ABB RobotStudio station: Solution_final_v2.rsstn

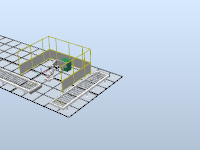
Station Solution1_1 (saved by RobotStudio 21.1.9393.1)
Controller Controlador1, task T_ROB1: task frame (RAPID world) sits at (-200, -1000, 0) mm in the station
Controller Controlador1
  mechanical unit ROB_1: IRB1600_6_120__02, 6 joints, base frame (0, 0, 0) mm
Layout (positions relative to the parent item):
  - IRB1600_6_120__02 [mechanism, from Robots\IRB1600_6_120_G_02.rslib] at (-200, -1000, 0) mm; joint values [0.1941, 0.1473, -0.2355, 0.1043, 1.3308, 0.4277] (rad or m)
  - RA_MTG4000_22 [mechanism, from Tools\Fronius_Robacta_MTG4000_22deg.rslib] at (621.28, -831.87, 948.02) mm, rotated rx 166.41 ry 14.43 rz 164.42 deg
  - Fence_740 [graphiccomponentgroup, from Equipment\Fence_740.rslib] at (2000, 225, 0) mm
    - Body 1 [part, from Equipment\Fence_740.rslib]
    - Body 2 [part, from Equipment\Fence_740.rslib]
  - Fence_740_2 [graphiccomponentgroup, from Equipment\Fence_740.rslib] at (2000, 925, 0) mm, rotated rx 0 ry 0 rz 90 deg
    - Body 1 [part, from Equipment\Fence_740.rslib]
    - Body 2 [part, from Equipment\Fence_740.rslib]
  - Fence_740_3 [graphiccomponentgroup, from Equipment\Fence_740.rslib] at (2000, -2940, 0) mm, rotated rx 0 ry 0 rz 90 deg
    - Body 1 [part, from Equipment\Fence_740.rslib]
    - Body 2 [part, from Equipment\Fence_740.rslib]
  - Fence_740_4 [graphiccomponentgroup, from Equipment\Fence_740.rslib] at (2000, -2240, 0) mm, rotated rx 0 ry 0 rz 180 deg
    - Body 1 [part, from Equipment\Fence_740.rslib]
    - Body 2 [part, from Equipment\Fence_740.rslib]
  - Fence_2500 [graphiccomponentgroup, from Equipment\Fence_2500.rslib] at (2000, 225, 0) mm, rotated rx 0 ry 0 rz 180 deg
    - Body 1 [part, from Equipment\Fence_2500.rslib]
    - Body 2 [part, from Equipment\Fence_2500.rslib]
  - Fence_2500_2 [graphiccomponentgroup, from Equipment\Fence_2500.rslib] at (1300, 925, 0) mm, rotated rx 0 ry 0 rz 90 deg
    - Body 1 [part, from Equipment\Fence_2500.rslib]
    - Body 2 [part, from Equipment\Fence_2500.rslib]
  - Fence_2500_3 [graphiccomponentgroup, from Equipment\Fence_2500.rslib] at (1300, -2940, 0) mm, rotated rx 0 ry 0 rz 90 deg
    - Body 1 [part, from Equipment\Fence_2500.rslib]
    - Body 2 [part, from Equipment\Fence_2500.rslib]
  - ConveyorControl_2 [smart component, from Components\ConveyorControl.rslib]
      properties: Conveyor=(none)
  - Process [smart component]
      signals: DI inicio, DI inicio2, DO sal_conv1, DO sal_conv2
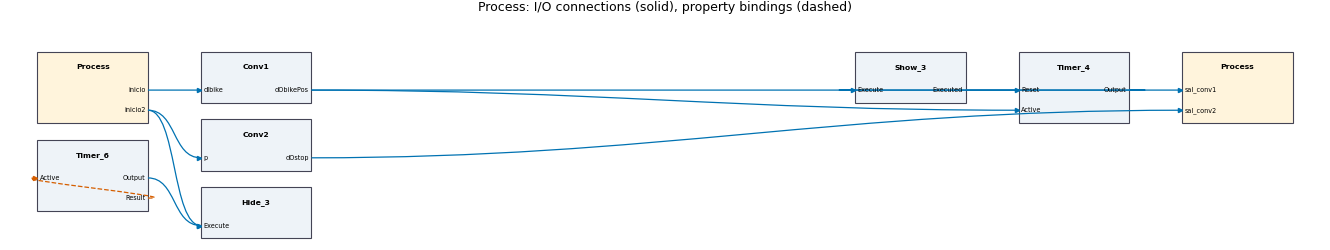
      connections:
        Timer_4.Output -> Show_3.Execute
        Show_3.Executed -> Timer_4.Reset
        Process.inicio -> Conv1.dIbike
        Conv1.dObikePos -> Timer_4.Active
        Timer_6.Output -> Hide_3.Execute
        Process.inicio2 -> Hide_3.Execute
        Conv1.dObikePos -> Process.sal_conv1
        Process.inicio2 -> Conv2.p
        Conv2.dOstop -> Process.sal_conv2
        Expression.Result => Timer_6.Active
    - Show_3 [smart component, from Components\Show.rslib]
        properties: Object=Bicycle Frame:1
    - Conv1 [smart component]
        signals: DI dIbike, DO dObikePos
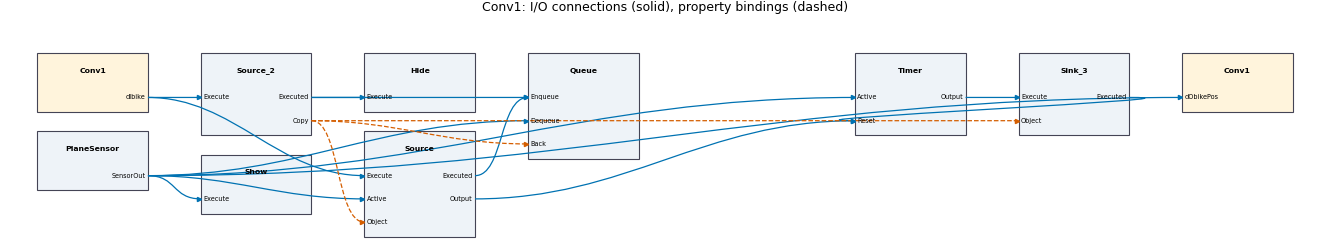
        connections:
          Conv1.dIbike -> Source.Execute
          Source.Executed -> Queue.Enqueue
          Conv1.dIbike -> Source_2.Execute
          Source_2.Executed -> Queue.Enqueue
          PlaneSensor.SensorOut -> Queue.Dequeue
          Source_2.Executed -> Hide.Execute
          PlaneSensor.SensorOut -> Show.Execute
          PlaneSensor.SensorOut -> Timer.Active
          Timer.Output -> Sink_3.Execute
          PlaneSensor.SensorOut -> Timer_5.Active
          Timer_5.Output -> Timer.Reset
          Sink_3.Executed -> Timer.Reset
          PlaneSensor.SensorOut -> Conv1.dObikePos
          Source_2.Copy => Queue.Back
          Source_2.Copy => Sink_2.Object
          Source_2.Copy => Sink_3.Object
      - 950_4800_h2 [part, from Equipment\Conveyor 950 4800 h2.rslib] at (2000, -3500, 0) mm, rotated rx 0 ry 0 rz 180 deg
      - Queue [smart component, from Components\Queue.rslib]
          properties: Back=(none); Front=(none); Queue={da4324a3-2cbe-466d-a78a-5e31958a6c5f};{e6e05bde-ee74-4659-88fe-c98839943faa};{f81fb27c-e148-4b64-9271-b941438183ca};{ce758764-b67b-4225-94dd-49e0e7ae394e}; NumberOfObjects=0
      - LinearMover [smart component, from Components\LinearMover.rslib]
          properties: Object=Queue; Direction=[-1 0 0]; Speed=0.5; Reference=Global; ReferenceObject=(none)
      - PlaneSensor [smart component, from Components\PlaneSensor.rslib]
          properties: Origin=[-2.65992 -3.5 0.435]; Axis1=[0 -0.91 0]; Axis2=[0 0 0.2]; SensedPart=(none)
        - _sensorPart_ [part]
      - Source_2 [smart component, from Components\Source.rslib]
          properties: Source=Bike; Copy=(none); Parent=(none); Position=[0 0 0]; Orientation=[0 0 0]; Transient=false; PhysicsBehavior=0
      - Show [smart component, from Components\Show.rslib]
          properties: Object=Bike
      - Hide [smart component, from Components\Hide.rslib]
          properties: Object=Bike
      - Sink_3 [smart component, from Components\Sink.rslib]
          properties: Object=(none)
      - Timer [smart component, from Components\Timer.rslib]
          properties: StartTime=3; Interval=3; Repeat=false; CurrentTime=0
    - Timer_4 [smart component, from Components\Timer.rslib]
        properties: StartTime=3; Interval=3; Repeat=false; CurrentTime=0
    - Conv2 [smart component]
        signals: DI p, DO dOstop
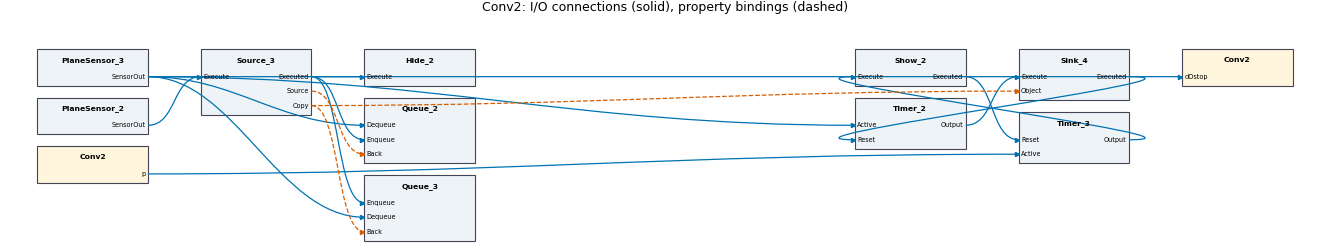
        connections:
          PlaneSensor_3.SensorOut -> Queue_2.Dequeue
          Source_3.Executed -> Queue_2.Enqueue
          Source_3.Executed -> Queue_3.Enqueue
          PlaneSensor_3.SensorOut -> Queue_3.Dequeue
          Source_3.Executed -> Hide_2.Execute
          PlaneSensor_3.SensorOut -> Timer_2.Active
          Timer_2.Output -> Sink_4.Execute
          Sink_4.Executed -> Timer_2.Reset
          PlaneSensor_2.SensorOut -> Source_3.Execute
          Timer_3.Output -> Show_2.Execute
          Show_2.Executed -> Timer_3.Reset
          Conv2.p -> Timer_3.Active
          PlaneSensor_3.SensorOut -> Conv2.dOstop
          Source_3.Source => Queue_2.Back
          Source_3.Copy => Queue_3.Back
          Source_3.Copy => Sink_4.Object
      - 950_4800_h2_3 [part, from Equipment\Conveyor 950 4800 h2.rslib] at (-1700, -1500, 0) mm, rotated rx 0 ry 0 rz 90 deg
      - Source_3 [smart component, from Components\Source.rslib]
          properties: Source=Bike2; Copy=Bike2_46; Parent=(none); Position=[0 0 0]; Orientation=[0 0 0]; Transient=false; PhysicsBehavior=0
      - LinearMover_2 [smart component, from Components\LinearMover.rslib]
          properties: Object=Queue_3; Direction=[0 1 0]; Speed=0.5; Reference=Global; ReferenceObject=(none)
      - PlaneSensor_2 [smart component, from Components\PlaneSensor.rslib]
          properties: Origin=[-2.61 -1.247316 0.435]; Axis1=[0.91 0 0]; Axis2=[0 0 0.2]; SensedPart=(none)
        - _sensorPart_ [part]
      - PlaneSensor_3 [smart component, from Components\PlaneSensor.rslib]
          properties: Origin=[-2.61 3.153624 0.435]; Axis1=[0.91 0 0]; Axis2=[0 0 0.2]; SensedPart=(none)
        - _sensorPart_ [part]
      - Hide_2 [smart component, from Components\Hide.rslib]
          properties: Object=Bike2
      - Show_2 [smart component, from Components\Show.rslib]
          properties: Object=Bike2
      - Queue_3 [smart component, from Components\Queue.rslib]
          properties: Back=Bike2_46; Front=Bike2_46; Queue={1f08c73b-8c5d-47c5-8fad-b47ddc3f47b2};{69fdafc0-c70e-498c-bd5d-4343ecce45a8};{ab0811c3-1ba0-43c0-b674-f4a10a17c4ae};{44498bd1-b295-4fc8-a058-8143949b90d9};{61c4f5f8-9c20-4886-aed5-0f792fba9fef};{207447c9-6041-471c-927b-d307d36bb852};{d11dc4f1-6705-4b2f-9a87-b3149d9034c5};{ffd23da9-bf60-4005-aac2-4753273c3d85};{c9eaf6c6-1d88-4ec3-ab1c-7dd69f2dac15}; NumberOfObjects=1
      - Sink_4 [smart component, from Components\Sink.rslib]
          properties: Object=Bike2_46
      - Timer_2 [smart component, from Components\Timer.rslib]
          properties: StartTime=3; Interval=3; Repeat=false; CurrentTime=0
      - Timer_3 [smart component, from Components\Timer.rslib]
          properties: StartTime=3; Interval=3; Repeat=true; CurrentTime=0
    - Hide_3 [smart component, from Components\Hide.rslib]
        properties: Object=Bicycle Frame:1
  - Bike [part]
  - Bike2 [part]
  - Soporte [smart component]
      signals: DI in_sop1, DI in_sop2, DI in_sop3, DO out_sop1, DO out_sop2, DO out_sop3
      connections:
        Soporte.in_sop1 -> JointMover.Execute
        Soporte.in_sop2 -> JointMover_2.Execute
        Soporte.in_sop3 -> JointMover_3.Execute
        JointMover_2.Executed -> Soporte.out_sop2
        JointMover_3.Executed -> Soporte.out_sop3
        JointMover.Executing -> Soporte.out_sop1
    - 2GDL_2 [mechanism, from Libraries\2GDL.rslib] at (1150, -1200, 0) mm, rotated rx 0 ry 0 rz -90 deg; joint values [0, 0] (rad or m)
    - JointMover [smart component, from Components\JointMover.rslib]
        properties: Mechanism=2GDL_2; Relative=false; Duration=2; J1=0; J2=0
    - JointMover_2 [smart component, from Components\JointMover.rslib]
        properties: Mechanism=2GDL_2; Relative=false; Duration=2; J1=0; J2=1.5707963267949
    - JointMover_3 [smart component, from Components\JointMover.rslib]
        properties: Mechanism=2GDL_2; Relative=false; Duration=2; J1=0; J2=3.14159265358979
  - Bike2_43 [part] at (0, 119076, 0) mm
  - Bike2_46 [part] at (0, 70188, 0) mm
Attachment: RA_MTG4000_22 is attached to IRB1600_6_120__02 / Link6
Station logic (signal -> signal, property => property):
  Soporte.out_sop1 -> Controlador1.in_so1
  Soporte.out_sop2 -> Controlador1.in_so2
  Soporte.out_sop3 -> Controlador1.in_so3
  Controlador1.out_so1 -> Soporte.in_sop1
  Controlador1.out_so2 -> Soporte.in_sop2
  Controlador1.out_so3 -> Soporte.in_sop3
  Process.sal_conv1 -> Controlador1.in_conv1
  Process.sal_conv2 -> Controlador1.in_conv2
  Controlador1.out_conv1 -> Process.inicio
  Controlador1.out_conv2 -> Process.inicio2
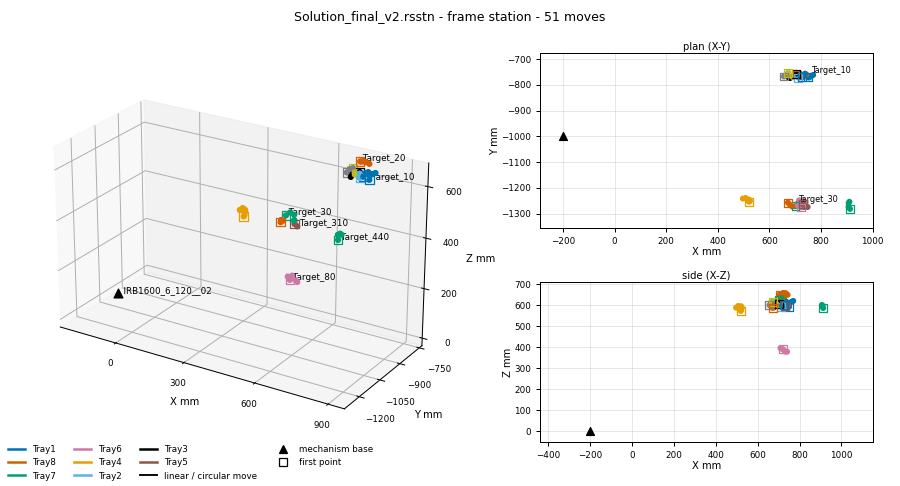
[picture p0: tool path of Solution_final_v2.rsstn in frame station, 51 of 51 moves have a stored position in this frame; points joined in program order, loops and branches not executed]
Targets, tools, work objects and paths stored in the station, written as RAPID:
! task T_ROB1
MODULE Module1
  PERS tooldata Weldgun:=[TRUE,[[20.31,0,363.689],[0.948464781,0,0.316882565,0]],[1,[0,0,1],[1,0,0,0],0,0,0]];
  CONST robtarget Target_10:=[[950.180013402,230.509872726,593.391104461],[0.01996439,-0.519361905,0.843066946,0.138212732],[-1,0,-1,0],[9E+09,9E+09,9E+09,9E+09,9E+09,9E+09]];
  CONST robtarget Target_10_2:=[[953.663168077,228.29744984,612.249682823],[0.033007773,0.167574443,-0.975918782,-0.135690173],[-1,0,-1,0],[9E+09,9E+09,9E+09,9E+09,9E+09,9E+09]];
  CONST robtarget Target_10_2_2:=[[961.689418242,232.938662049,617.331587375],[0.009863037,-0.321024311,0.935655547,0.146269649],[0,0,-1,0],[9E+09,9E+09,9E+09,9E+09,9E+09,9E+09]];
  CONST robtarget Target_10_2_2_2:=[[970.054312191,238.235263505,621.336954731],[0.065377578,-0.311777181,0.933420781,0.16506486],[-1,0,-1,0],[9E+09,9E+09,9E+09,9E+09,9E+09,9E+09]];
  CONST robtarget Target_20:=[[905.762920651,240.030211699,651.609928361],[0.228486899,-0.080722826,0.930320129,0.275285344],[0,0,0,0],[9E+09,9E+09,9E+09,9E+09,9E+09,9E+09]];
  CONST robtarget Target_20_2:=[[912.116723412,238.074295519,653.417444244],[0.226392928,-0.086421523,0.923131727,0.298505237],[0,0,-1,0],[9E+09,9E+09,9E+09,9E+09,9E+09,9E+09]];
  CONST robtarget Target_20_2_2:=[[922.807470131,229.791716616,659.467831703],[0.154916171,-0.109064049,0.937777652,0.290996717],[-1,0,-1,0],[9E+09,9E+09,9E+09,9E+09,9E+09,9E+09]];
  CONST robtarget Target_20_2_2_2:=[[926.560901787,231.240903084,659.344619966],[0.015873837,0.159510477,-0.950354652,-0.26670295],[-1,0,-1,0],[9E+09,9E+09,9E+09,9E+09,9E+09,9E+09]];
  CONST robtarget Target_20_2_2_2_2:=[[935.042483171,230.884165583,657.882908466],[0.134813361,0.177010196,-0.91890316,-0.325744886],[-1,0,-1,0],[9E+09,9E+09,9E+09,9E+09,9E+09,9E+09]];
  CONST robtarget Target_20_2_2_2_2_2:=[[943.210532645,240.444228342,650.282226312],[0.301906779,0.213670219,-0.851210168,-0.372342026],[-1,0,-1,0],[9E+09,9E+09,9E+09,9E+09,9E+09,9E+09]];
  CONST robtarget Target_30:=[[901.556015815,-270.162237253,625.680850338],[0.197428015,0.10740669,0.956069337,-0.188195126],[0,0,0,0],[9E+09,9E+09,9E+09,9E+09,9E+09,9E+09]];
  CONST robtarget Target_40:=[[911.417050152,-258.539768811,634.430430873],[0.220426883,0.020508221,0.956040611,-0.192296001],[0,0,0,0],[9E+09,9E+09,9E+09,9E+09,9E+09,9E+09]];
  CONST robtarget Target_50:=[[927.223704569,-259.545949624,629.928676022],[0.077790476,0.047659901,-0.973242925,0.210891877],[0,0,0,0],[9E+09,9E+09,9E+09,9E+09,9E+09,9E+09]];
  CONST robtarget Target_60:=[[935.783661558,-273.343346853,616.363371194],[0.373650363,-0.169699504,-0.879731127,0.240126278],[0,0,0,0],[9E+09,9E+09,9E+09,9E+09,9E+09,9E+09]];
  CONST robtarget Target_70:=[[935.801859981,-274.112324453,615.600810011],[0.367877976,-0.102265478,-0.905499304,0.185144746],[0,0,0,0],[9E+09,9E+09,9E+09,9E+09,9E+09,9E+09]];
  CONST robtarget Target_80:=[[922.550948175,-275.513815971,390.102644127],[0.101847243,0.339270429,0.880891165,0.313932271],[0,0,0,0],[9E+09,9E+09,9E+09,9E+09,9E+09,9E+09]];
  CONST robtarget Target_90:=[[908.919438616,-267.012467724,396.003979358],[0.140986165,0.2630963,0.920921902,0.25061143],[0,0,0,0],[9E+09,9E+09,9E+09,9E+09,9E+09,9E+09]];
  CONST robtarget Target_110:=[[915.336985705,-247.556480637,393.478283582],[0.180039373,0.336799833,0.91219813,0.148479858],[0,0,0,0],[9E+09,9E+09,9E+09,9E+09,9E+09,9E+09]];
  CONST robtarget Target_170:=[[707.852315504,-238.649710951,597.523713075],[0.072970374,0.005434554,0.928587731,-0.363827728],[0,0,0,0],[9E+09,9E+09,9E+09,9E+09,9E+09,9E+09]];
  CONST robtarget Target_180:=[[721.007297904,-244.597864758,596.203274989],[0.277568826,-0.191544592,-0.908750875,0.245841539],[0,0,0,0],[9E+09,9E+09,9E+09,9E+09,9E+09,9E+09]];
  CONST robtarget Target_190:=[[724.403295258,-249.007768841,590.910196548],[0.017591206,-0.2639641,-0.951251292,0.158538588],[0,0,0,0],[9E+09,9E+09,9E+09,9E+09,9E+09,9E+09]];
  CONST robtarget Target_190_2:=[[723.102759435,-252.252697135,580.374954479],[0.271606911,-0.330293045,-0.838598066,0.337475146],[0,-1,0,0],[9E+09,9E+09,9E+09,9E+09,9E+09,9E+09]];
  CONST robtarget Target_190_2_2:=[[720.242148182,-252.666792281,573.887180235],[0.335060979,-0.265702747,-0.748744935,0.506475284],[0,-1,0,0],[9E+09,9E+09,9E+09,9E+09,9E+09,9E+09]];
  CONST robtarget Target_200:=[[912.737551752,227.954555454,593.425678044],[0.091839012,-0.179736425,-0.96617993,-0.160489117],[0,0,0,0],[9E+09,9E+09,9E+09,9E+09,9E+09,9E+09]];
  CONST robtarget Target_210:=[[907.911596267,235.490164986,606.563398786],[0.24680063,0.002115266,-0.963219889,-0.106265801],[0,0,0,0],[9E+09,9E+09,9E+09,9E+09,9E+09,9E+09]];
  CONST robtarget Target_220:=[[902.907851772,243.466885632,608.834913969],[0.000730197,0.162791926,-0.986591136,-0.011669883],[0,0,0,0],[9E+09,9E+09,9E+09,9E+09,9E+09,9E+09]];
  CONST robtarget Target_230:=[[902.907851772,243.466885632,608.834913969],[0.047897344,-0.306115236,0.950411946,0.026766386],[0,0,0,0],[9E+09,9E+09,9E+09,9E+09,9E+09,9E+09]];
  CONST robtarget Target_240:=[[882.23790733,227.202137761,600.639163926],[0.196683297,-0.050586157,0.908908918,0.364199533],[0,0,0,0],[9E+09,9E+09,9E+09,9E+09,9E+09,9E+09]];
  CONST robtarget Target_240_2:=[[876.573137523,226.169639566,590.457482001],[0.243900527,-0.068597657,0.886317922,0.387617642],[0,0,0,0],[9E+09,9E+09,9E+09,9E+09,9E+09,9E+09]];
  CONST robtarget Target_250:=[[697.382168192,-241.204197142,589.059929206],[0.284999056,0.337553205,0.869802576,-0.219719939],[0,-2,1,0],[9E+09,9E+09,9E+09,9E+09,9E+09,9E+09]];
  CONST robtarget Target_110_2:=[[930.843064777,-249.326046664,379.537564288],[0.152197256,-0.012389746,0.972056809,-0.178292037],[-1,-1,0,0],[9E+09,9E+09,9E+09,9E+09,9E+09,9E+09]];
  CONST robtarget Target_110_2_2:=[[940.589509157,-255.917178356,379.084460502],[0.06036507,-0.012599268,0.99290881,-0.101633709],[-1,0,-1,0],[9E+09,9E+09,9E+09,9E+09,9E+09,9E+09]];
  CONST robtarget Target_290:=[[931.040939153,-262.788731504,597.974884508],[0.127428962,0.031592152,0.910868387,-0.391257686],[0,0,0,0],[9E+09,9E+09,9E+09,9E+09,9E+09,9E+09]];
  CONST robtarget Target_300:=[[932.336369047,-264.703643694,610.813063224],[0.220344948,0.177840656,0.956824655,0.065630673],[0,0,0,0],[9E+09,9E+09,9E+09,9E+09,9E+09,9E+09]];
  CONST robtarget Target_310:=[[948.397176267,-273.682088466,596.848598959],[0.012121441,-0.133462629,-0.98955513,0.05311725],[0,0,0,0],[9E+09,9E+09,9E+09,9E+09,9E+09,9E+09]];
  CONST robtarget Target_320:=[[856.630830609,232.178913763,601.139433385],[0.279369762,-0.65025277,-0.262269636,-0.656001913],[0,0,0,0],[9E+09,9E+09,9E+09,9E+09,9E+09,9E+09]];
  CONST robtarget Target_330:=[[863.969144353,238.19760156,613.755907331],[0.06759041,-0.894729801,-0.3229049,-0.301035787],[0,0,0,0],[9E+09,9E+09,9E+09,9E+09,9E+09,9E+09]];
  CONST robtarget Target_340:=[[873.11969206,246.05387669,616.468662664],[0.104899831,-0.520682064,0.84418492,0.072374273],[0,0,0,0],[9E+09,9E+09,9E+09,9E+09,9E+09,9E+09]];
  CONST robtarget Target_350:=[[873.11969206,246.05387669,616.468662664],[0.047936139,0.452328602,-0.88307423,-0.11524264],[0,0,0,0],[9E+09,9E+09,9E+09,9E+09,9E+09,9E+09]];
  CONST robtarget Target_360:=[[888.670577795,232.264868573,608.080812591],[0.04172614,0.21845991,-0.933015424,-0.282871729],[0,0,0,0],[9E+09,9E+09,9E+09,9E+09,9E+09,9E+09]];
  CONST robtarget Target_370:=[[890.687396471,230.61872251,601.040016664],[0.014668168,0.105360192,-0.954769294,-0.277668275],[0,0,0,0],[9E+09,9E+09,9E+09,9E+09,9E+09,9E+09]];
  CONST robtarget Target_380:=[[926.311547498,228.986717421,600.936023904],[0.118885249,-0.400714438,0.901490949,0.112286715],[0,0,0,0],[9E+09,9E+09,9E+09,9E+09,9E+09,9E+09]];
  CONST robtarget Target_390:=[[932.183277776,235.803444297,614.040602566],[0.175749755,-0.390650962,0.893386243,0.135517047],[0,0,0,0],[9E+09,9E+09,9E+09,9E+09,9E+09,9E+09]];
  CONST robtarget Target_400:=[[938.18034038,243.073333825,616.278739923],[0.00545867,-0.488935138,0.872226861,0.011529805],[0,0,0,0],[9E+09,9E+09,9E+09,9E+09,9E+09,9E+09]];
  CONST robtarget Target_410:=[[872.089272642,-256.677280849,588.666367493],[0.317356463,0.25138082,0.908911492,0.099862199],[0,0,0,0],[9E+09,9E+09,9E+09,9E+09,9E+09,9E+09]];
  CONST robtarget Target_420:=[[878.984440574,-264.335321237,600.935417335],[0.220825711,0.253575524,0.935479268,0.108692222],[0,0,0,0],[9E+09,9E+09,9E+09,9E+09,9E+09,9E+09]];
  CONST robtarget Target_430:=[[888.966656062,-271.907970792,603.185354603],[0.042205837,0.32810717,-0.943319414,-0.026698968],[0,0,0,0],[9E+09,9E+09,9E+09,9E+09,9E+09,9E+09]];
  CONST robtarget Target_440:=[[1112.804158472,-281.213807605,587.619751686],[0.177269991,0.058325125,0.982419704,-0.005005475],[0,0,0,0],[9E+09,9E+09,9E+09,9E+09,9E+09,9E+09]];
  CONST robtarget Target_450:=[[1107.052335394,-272.939547734,601.503437689],[0.244055824,-0.042649205,0.968616185,0.020012176],[0,0,0,0],[9E+09,9E+09,9E+09,9E+09,9E+09,9E+09]];
  CONST robtarget Target_460:=[[1107.381164317,-258.472924707,600.755996436],[0.168215177,-0.123924584,0.948996575,-0.236118303],[0,0,0,0],[9E+09,9E+09,9E+09,9E+09,9E+09,9E+09]];
  CONST robtarget Target_470:=[[1110.195892968,-253.412409389,595.702325754],[0.123463154,-0.227579271,0.952556976,-0.159999163],[0,0,0,0],[9E+09,9E+09,9E+09,9E+09,9E+09,9E+09]];
  PROC Tray1()
    MoveL Target_10,v1000,z100,Weldgun\WObj:=wobj0;
    MoveL Target_10_2,v1000,z100,Weldgun\WObj:=wobj0;
    MoveL Target_10_2_2,v1000,z100,Weldgun\WObj:=wobj0;
    MoveL Target_10_2_2_2,v1000,z100,Weldgun\WObj:=wobj0;
  ENDPROC
  PROC Tray8()
    MoveL Target_20,v1000,z100,Weldgun\WObj:=wobj0;
    MoveL Target_20_2,v1000,z100,Weldgun\WObj:=wobj0;
    MoveL Target_20_2_2,v1000,z100,Weldgun\WObj:=wobj0;
    MoveL Target_20_2_2_2,v1000,z100,Weldgun\WObj:=wobj0;
    MoveL Target_20_2_2_2_2,v1000,z100,Weldgun\WObj:=wobj0;
    MoveL Target_20_2_2_2_2_2,v1000,z100,Weldgun\WObj:=wobj0;
  ENDPROC
  PROC Tray7()
    MoveL Target_30,v1000,z100,Weldgun\WObj:=wobj0;
    MoveL Target_40,v1000,z100,Weldgun\WObj:=wobj0;
    MoveL Target_50,v1000,z100,Weldgun\WObj:=wobj0;
    MoveL Target_60,v1000,z100,Weldgun\WObj:=wobj0;
    MoveL Target_70,v1000,z100,Weldgun\WObj:=wobj0;
  ENDPROC
  PROC Tray6()
    MoveL Target_80,v1000,z100,Weldgun\WObj:=wobj0;
    MoveL Target_90,v1000,z100,Weldgun\WObj:=wobj0;
    MoveL Target_110,v1000,z100,Weldgun\WObj:=wobj0;
    MoveL Target_110_2,v1000,z100,Weldgun\WObj:=wobj0;
    MoveL Target_110_2_2,v1000,z100,Weldgun\WObj:=wobj0;
  ENDPROC
  PROC Tray4()
    MoveL Target_190_2_2,v1000,z100,Weldgun\WObj:=wobj0;
    MoveL Target_190_2,v1000,z100,Weldgun\WObj:=wobj0;
    MoveL Target_190,v1000,z100,Weldgun\WObj:=wobj0;
    MoveL Target_180,v1000,z100,Weldgun\WObj:=wobj0;
    MoveL Target_170,v1000,z100,Weldgun\WObj:=wobj0;
    MoveL Target_250,v1000,z100,Weldgun\WObj:=wobj0;
  ENDPROC
  PROC Tray2()
    MoveL Target_200,v1000,z100,Weldgun\WObj:=wobj0;
    MoveL Target_210,v1000,z100,Weldgun\WObj:=wobj0;
    MoveL Target_220,v1000,z100,Weldgun\WObj:=wobj0;
  ENDPROC
  PROC Tray3()
    MoveL Target_230,v1000,z100,Weldgun\WObj:=wobj0;
    MoveL Target_240,v1000,z100,Weldgun\WObj:=wobj0;
    MoveL Target_240_2,v1000,z100,Weldgun\WObj:=wobj0;
  ENDPROC
  PROC Tray5()
    MoveL Target_290,v1000,z100,Weldgun\WObj:=wobj0;
    MoveL Target_300,v1000,z100,Weldgun\WObj:=wobj0;
    MoveL Target_310,v1000,z100,Weldgun\WObj:=wobj0;
  ENDPROC
  PROC Tray9()
    MoveL Target_320,v1000,z100,Weldgun\WObj:=wobj0;
    MoveL Target_330,v1000,z100,Weldgun\WObj:=wobj0;
    MoveL Target_340,v1000,z100,Weldgun\WObj:=wobj0;
  ENDPROC
  PROC Tray10()
    MoveL Target_350,v1000,z100,Weldgun\WObj:=wobj0;
    MoveL Target_360,v1000,z100,Weldgun\WObj:=wobj0;
    MoveL Target_370,v1000,z100,Weldgun\WObj:=wobj0;
  ENDPROC
  PROC Tray11()
    MoveL Target_380,v1000,z100,Weldgun\WObj:=wobj0;
    MoveL Target_390,v1000,z100,Weldgun\WObj:=wobj0;
    MoveL Target_400,v1000,z100,Weldgun\WObj:=wobj0;
  ENDPROC
  PROC Tray12()
    MoveL Target_410,v1000,z100,Weldgun\WObj:=wobj0;
    MoveL Target_420,v1000,z100,Weldgun\WObj:=wobj0;
    MoveL Target_430,v1000,z100,Weldgun\WObj:=wobj0;
  ENDPROC
  PROC Tray13()
    MoveL Target_440,v1000,z100,Weldgun\WObj:=wobj0;
    MoveL Target_450,v1000,z100,Weldgun\WObj:=wobj0;
    MoveL Target_460,v1000,z100,Weldgun\WObj:=wobj0;
    MoveL Target_470,v1000,z100,Weldgun\WObj:=wobj0;
  ENDPROC
ENDMODULE

